FUNCTION_BLOCK FB_PowerAll
VAR_INPUT
	Enable : BOOL;
END_VAR
VAR_OUTPUT
	Status	: BOOL;
	Error	: BOOL;
END_VAR
VAR
	fbPower	: ARRAY[1..cAxesCount] OF MC_Power;
	i		: UINT;
END_VAR

Status	:= TRUE;
Error	:= FALSE;

FOR i := 1 TO cAxesCount DO
	fbPower[i](Axis				:= stAxis[i],
				Enable			:= Enable,
				Enable_Positive	:= Enable,
				Enable_Negative	:= Enable);

	Status	:= Status AND fbPower[i].Status;
	Error	:= Error OR fbPower[i].Error;
END_FOR

END_FUNCTION_BLOCK

(* stored: Version 1.1.0.1, ProductVersion 3.1.4024.12
   POU FB_PowerAll: Id {d3e6d2d4-b215-4a84-8022-bf06b4a82234}, SpecialFunc None *)
